(* CoDeSys 2.3.9.47 project: 2floor_2016-05-20.pr6 *)
(* Author: Yurko Shybaigolova *)
(* Libraries: TcAdsBC.lb6 5.7.02 11:03:02, standard.lb6 5.6.98 11:03:02, PlcSystemBC.lb6 21.3.01 11:03:02, TcPlcUtilitiesBC.lb6 13.5.05 11:19:40, TcBABasicBC.lb6 22.7.15 15:46:36 *)

(* Global variable list: main *)
VAR_GLOBAL
(*ADS*)
	ads_adr1: STRING:='10.0.5.61.1.1';
	ads_adr2: STRING:='10.0.5.62.1.1';
	ads_adr3: STRING:='10.0.5.63.1.1';

	write_ads: ADSWRITE;
	close_ads:ADSCLOSE;
	read_ads1: ADSREADEX;
	read_ads3: ADSREADEX;

	data1floor: ARRAY[0..4] OF BYTE;
	data1floor_prev: ARRAY[0..4] OF BYTE;
	data3floor: ARRAY[0..200] OF BYTE;
	data3floor_prev: ARRAY[0..200] OF BYTE;

	m_fancoil_kabinet_low 	AT%MX300.0: BOOL;
	m_fancoil_kabinet_med 	AT%MX300.1: BOOL;
	m_fancoil_kabinet_high 	AT%MX300.2: BOOL;
	m_fancoil_kino_low 		AT%MX300.3: BOOL;
	m_fancoil_kino_med 	AT%MX300.4: BOOL;
	m_fancoil_kino_high		AT%MX300.5: BOOL;

	tepla_pidloga_kabinet	AT%MX301.0:BOOL;
	tepla_pidloga_studio		AT%MX301.1:BOOL;

	m_klapan_kabinet		AT%MW302: WORD;


	m_klapan_kino			AT%MW304: WORD;

	sw_tambur3_2			AT%MX306.0:BOOL;
	bDarkOutside			AT%MX306.1:BOOL;
	bT_out_sign				AT%MX306.7:BOOL;

	eib_kabinet_shtory			AT%MX307.0:BOOL;
	eib_kabinet_tul				AT%MX307.1:BOOL;
	t_out3					AT%MB308:BYTE;
	t_out:REAL;
	iHour					AT%MB309:BYTE;
	iMinute					AT%MB310:BYTE;
	lights					AT%MB312:DWORD;

	eib_kino_shtory_move			AT%MX316.0:BOOL;
	eib_kino_tul_move				AT%MX316.1:BOOL;
	eib_kabinet_shtory_move		AT%MX316.2:BOOL;
	eib_kabinet_tul_move			AT%MX316.3:BOOL;
	eib_kino_shtory_position			AT%MB317	:BYTE;
	eib_kino_tul_position				AT%MB318	:BYTE;
	eib_kabinet_shtory_position		AT%MB319	:BYTE;
	eib_kabinet_tul_position			AT%MB320	:BYTE;


	eib_balkon_peryla 				AT%MX400.0:BOOL;
	eib_kino_l						AT%MX400.1:BOOL;
	eib_balkon_bra					AT%MX400.2:BOOL;
	eib_kabinet_balkon_l			AT%MX400.3:BOOL;
	eib_balkon						AT%MX400.4:BOOL;
	eib_korydor1					AT%MX400.5:BOOL;
	eib_kino_bra					AT%MX400.6:BOOL;
(*	eib_korydor2					AT%MX400.7:BOOL;
*)	eib_studio_pidsvitka				AT%MX401.0:BOOL;
	eib_skhody2_3					AT%MX401.1:BOOL;
	eib_studio_l						AT%MX401.2:BOOL;
(*	eib_kabinet_pidsvitka_kolo		AT%MX401.3:BOOL;
*)	eib_kabinet_svitlo				AT%MX401.4:BOOL;
	eib_kabinet_kobra				AT%MX401.5:BOOL;
	eib_tambur_l					AT%MX401.6:BOOL;
	eib_stend						AT%MX401.7:BOOL;
	eib_skhody_peryla				AT%MX402.0:BOOL;




	sw_tambur1_2			AT%MX100.0:BOOL;
	sw_vhid2				AT%MX100.1:BOOL;
	moove_kino				AT%MX101.0:BOOL;
	moove_skhody1_2		AT%MX101.1:BOOL;
	moove_studio			AT%MX101.2:BOOL;
	moove_kabinet			AT%MX101.3:BOOL;
	sw_tambur1_3_long		AT%MX101.4:BOOL;


	fbKino1_sw: FB_ShortLongClick;		(*processor for left button of the switch near the door in home cinema *)
END_VAR

(* Global variable list: physical *)
VAR_GLOBAL
(*	din1_1	AT %IX52.0:	BOOL;
	din1_2	AT %IX52.1:	BOOL;
	din1_3	AT %IX52.2:	BOOL;
	din1_4	AT %IX52.3:	BOOL;
	din1_5	AT %IX52.4:	BOOL;
	din1_6	AT %IX52.5:	BOOL;
	din1_7	AT %IX52.6:	BOOL;
	din1_8	AT %IX52.7:	BOOL;
	din2_1	AT %IX53.0:	BOOL;
	din2_2	AT %IX53.1:	BOOL;
	din2_3	AT %IX53.2:	BOOL;
	din2_4	AT %IX53.3:	BOOL;
	din2_5	AT %IX53.4:	BOOL;
	din2_6	AT %IX53.5:	BOOL;
	din2_7	AT %IX53.6:	BOOL;
	din2_8	AT %IX53.7:	BOOL;
*)

	sw_kino_balkon				AT %IX54.0:	BOOL;
	sw_tambur2_1				AT %IX54.1:	BOOL;
	sw_kino1					AT %IX54.2:	BOOL;
	sw_korydor					AT %IX54.3:	BOOL;
	sw_kino2					AT %IX54.4:	BOOL;
	sw_studio1					AT %IX54.5:	BOOL;
	sw_tambur2_2				AT %IX54.6:	BOOL;
	sw_studio2					AT %IX54.7:	BOOL;
	sw_kabinet1				AT %IX55.0:	BOOL;
(*	din4_2	AT %IX55.1:	BOOL;
*)	sw_kabinet2				AT %IX55.2:	BOOL;
	sw_kabinet2_1				AT %IX55.3:	BOOL;
	sw_kabinet_balkon			AT %IX55.4:	BOOL;
	sw_kabinet2_2				AT %IX55.5:	BOOL;
	sw_tambur3					AT %IX55.6:	BOOL;
(*	din4_8	AT %IX55.7:	BOOL;
*)

	balkon_peryla				AT %QX52.0:	BOOL;
	kino_l						AT %QX52.1:	BOOL;
	balkon_bra					AT %QX52.2:	BOOL;
	kabinet_balkon_l			AT %QX52.3:	BOOL;
	balkon						AT %QX52.4:	BOOL;
	korydor1					AT %QX52.5:	BOOL;
	kino_bra					AT %QX52.6:	BOOL;
	korydor2					AT %QX52.7:	BOOL;
	studio_pidsvitka 				AT %QX53.0:	BOOL;
	skhody2_3					AT %QX53.1:	BOOL;
	studio_l						AT %QX53.2:	BOOL;
	kabinet_pidsvitka_kolo		AT %QX53.3:	BOOL;
	kabinet_svitlo				AT %QX53.4:	BOOL;
	kabinet_kobra 				AT %QX53.5:	BOOL;
	tambur_l					AT %QX53.6:	BOOL;
	stend						AT %QX53.7:	BOOL;
	collector_kabinet1			AT %QX54.0:	BOOL;
	fancoil_kabinet_low			AT %QX54.1:	BOOL;
	collector_kabinet2			AT %QX54.2:	BOOL;
	fancoil_kabinet_med			AT %QX54.3:	BOOL;
	collector_studio1			AT %QX54.4:	BOOL;
	fancoil_kabinet_high			AT %QX54.5:	BOOL;
	collector_studio2			AT %QX54.6:	BOOL;
	fancoil_kino_low				AT %QX54.7:	BOOL;
	fancoil_kino_med			AT %QX55.0:	BOOL;
(*	dout4_2	AT %QX55.1:	BOOL;
*)	fancoil_kino_high			AT %QX55.2:	BOOL;
	skhody_peryla				AT %QX55.3:	BOOL;
(*	dout4_5	AT %QX55.4:	BOOL;
	dout4_6	AT %QX55.5:	BOOL;
	dout4_7	AT %QX55.6:	BOOL;
	dout4_8	AT %QX55.7:	BOOL;
*)	kino_tul_open				AT %QX56.0:	BOOL;
	kabinet_tul_close 			AT %QX56.1:	BOOL;
	kino_tul_close 				AT %QX56.2:	BOOL;
	kabinet_tul_open			AT %QX56.3:	BOOL;
	kino_shtory_open			AT %QX56.4:	BOOL;
	kabinet_shtory_open			AT %QX56.5:	BOOL;
	kino_shtory_close			AT %QX56.6:	BOOL;
	kabinet_shtory_close		AT %QX56.7:	BOOL;


	klapan_kino 				AT %QB2:	INT;
	klapan_kabinet				AT %QB6:	INT; (*0-opened, 16#7fff - closed*)

	temp_kabinet				AT %IB18:	INT;
	temp_studio		 			AT %IB26:	INT;


	Term_12_KL3228_4_1_State			AT %IB16:	USINT;

	Term_12_KL3228_4_1_Ctrl				AT %QB16:	USINT;
	Term_12_KL3228_4_1_Data_Out		AT %QB18:	INT;
	Term_12_KL3228_4_2_State			AT %IB20:	USINT;
	Term_12_KL3228_4_2_Data_In			AT %IB22:	INT;
	Term_12_KL3228_4_2_Ctrl				AT %QB20:	USINT;
	Term_12_KL3228_4_2_Data_Out		AT %QB22:	INT;
	Term_12_KL3228_4_3_State			AT %IB24:	USINT;

	Term_12_KL3228_4_3_Ctrl				AT %QB24:	USINT;
	Term_12_KL3228_4_3_Data_Out		AT %QB26:	INT;
	Term_12_KL3228_4_4_State			AT %IB28:	USINT;
	Term_12_KL3228_4_4_Data_In			AT %IB30:	INT;
	Term_12_KL3228_4_4_Ctrl				AT %QB28:	USINT;
	Term_12_KL3228_4_4_Data_Out		AT %QB30:	INT;
	Term_13_KL3228_4_1_State			AT %IB32:	USINT;
	Term_13_KL3228_4_1_Data_In			AT %IB34:	INT;
	Term_13_KL3228_4_1_Ctrl				AT %QB32:	USINT;
	Term_13_KL3228_4_1_Data_Out		AT %QB34:	INT;
	Term_13_KL3228_4_2_State			AT %IB36:	USINT;
	Term_13_KL3228_4_2_Data_In			AT %IB38:	INT;
	Term_13_KL3228_4_2_Ctrl				AT %QB36:	USINT;
	Term_13_KL3228_4_2_Data_Out		AT %QB38:	INT;
	Term_13_KL3228_4_3_State			AT %IB40:	USINT;
	Term_13_KL3228_4_3_Data_In			AT %IB42:	INT;
	Term_13_KL3228_4_3_Ctrl				AT %QB40:	USINT;
	Term_13_KL3228_4_3_Data_Out		AT %QB42:	INT;
	Term_13_KL3228_4_4_State			AT %IB44:	USINT;
	Term_13_KL3228_4_4_Data_In			AT %IB46:	INT;
	Term_13_KL3228_4_4_Ctrl				AT %QB44:	USINT;
	Term_13_KL3228_4_4_Data_Out		AT %QB46:	INT;
	Term_14_KL2761_State					AT %IB48:	USINT;
	kino_bra_state							AT %IB50:	INT;
	Term_14_KL2761_Ctrl					AT %QB48:	USINT;
	kino_bra_ctrl							AT %QB50:	INT;



END_VAR

(* POU MAIN, ST *)
PROGRAM MAIN
VAR

END_VAR
Light;
heat;
ADS1_write;
ADS3_write;
ADS_Communication;
END_PROGRAM

(* POU Light, CFC *)
PROGRAM Light
VAR
	longPressDelay: TIME:=t#500ms;
	lightDuration:INT:=120;




	fbKino_l							: FB_Light;						(*fb for home cinema mainlight switching*)
	fbKino_bra						: FB_Dimmer1SwitchEco;		(*fb for home cinema bra dimming*)
	fbKino2_sw						: FB_ShortLongClick;			(*processor for right button of the switch near the door in home cinema *)
	fbKino_bra_switching			: FB_Light;						(*fb for generating ON and OFF signals for 2SwitchDimmer fb*)
	fbKabinet_balkon				: FB_Light;		(*fb for balkony light switching in Oleg's cabinet*)
	fbKino_balkon					: FB_Light;		(*fb for switching balcony light in home cinema
			*)
	fbKabinet_l						: FB_Light;		(*fb for kabinet main light switching*)
	fbKabinet_kobra					: FB_Light;		(*fb for kabinet "cobra light" switching*)
	fStudio_l						: FB_Light;		(*fb for studio main light switching*)
	fStudio_pidsvitka				: FB_Light;		(*fb for studio  secondary light switching*)
	fbKorydor_l						: FB_Light;		(*fb for corridor light switching *)
	fbStend							: FB_Light;		(*fb for climbing wall light switching*)
	fbSkhody2_3					: FB_Light;		(*fb for stairs to the 3rd floor light switching*)

	fbKabinet1_sw: FB_ShortLongClick;				(*processor for left button of the kabinet switch near the door*)
	fbKabinet2_sw: FB_ShortLongClick;				(*processor for right button of the kabinet switch near the door*)
	fbKabinetShtory: FB_VenetianBlindEx1Switch;		(*fb for shtory control in kabinet*)

	fbKabinetShtorySwitching: FB_Light;				(*fb for ON and OFF signals generation for shtory control*)

	fbKabinetTulSwitching: FB_Light;					(*fb for ON and OFF signals generation for tul control*)
	fbKabinetTul: FB_VenetianBlindEx1Switch;		(*fb for ON and OFF signals generation for tul control*)

	fbKinoShtory: FB_VenetianBlindEx1Switch;
	kino_shtory_up_trigger: R_TRIG;
	kino_shtory_down_trigger: R_TRIG;

	kino_shtoryActualPosition: 	USINT;				(*position of the kino shtory*)
	kabinet_tulActualPosition: 	USINT;				(*position of the kabinet tul*)
	kabinet_shtoryActualPosition: USINT;				(*position of the kabinet shtory*)
	kino_tulActualPosition: 		USINT;					(*position of the kabinet shtory*)

	fbKinoTul: FB_VenetianBlindEx1Switch;
END_VAR
VAR CONSTANT
	msecMultiplier: DINT := 1000;
END_VAR
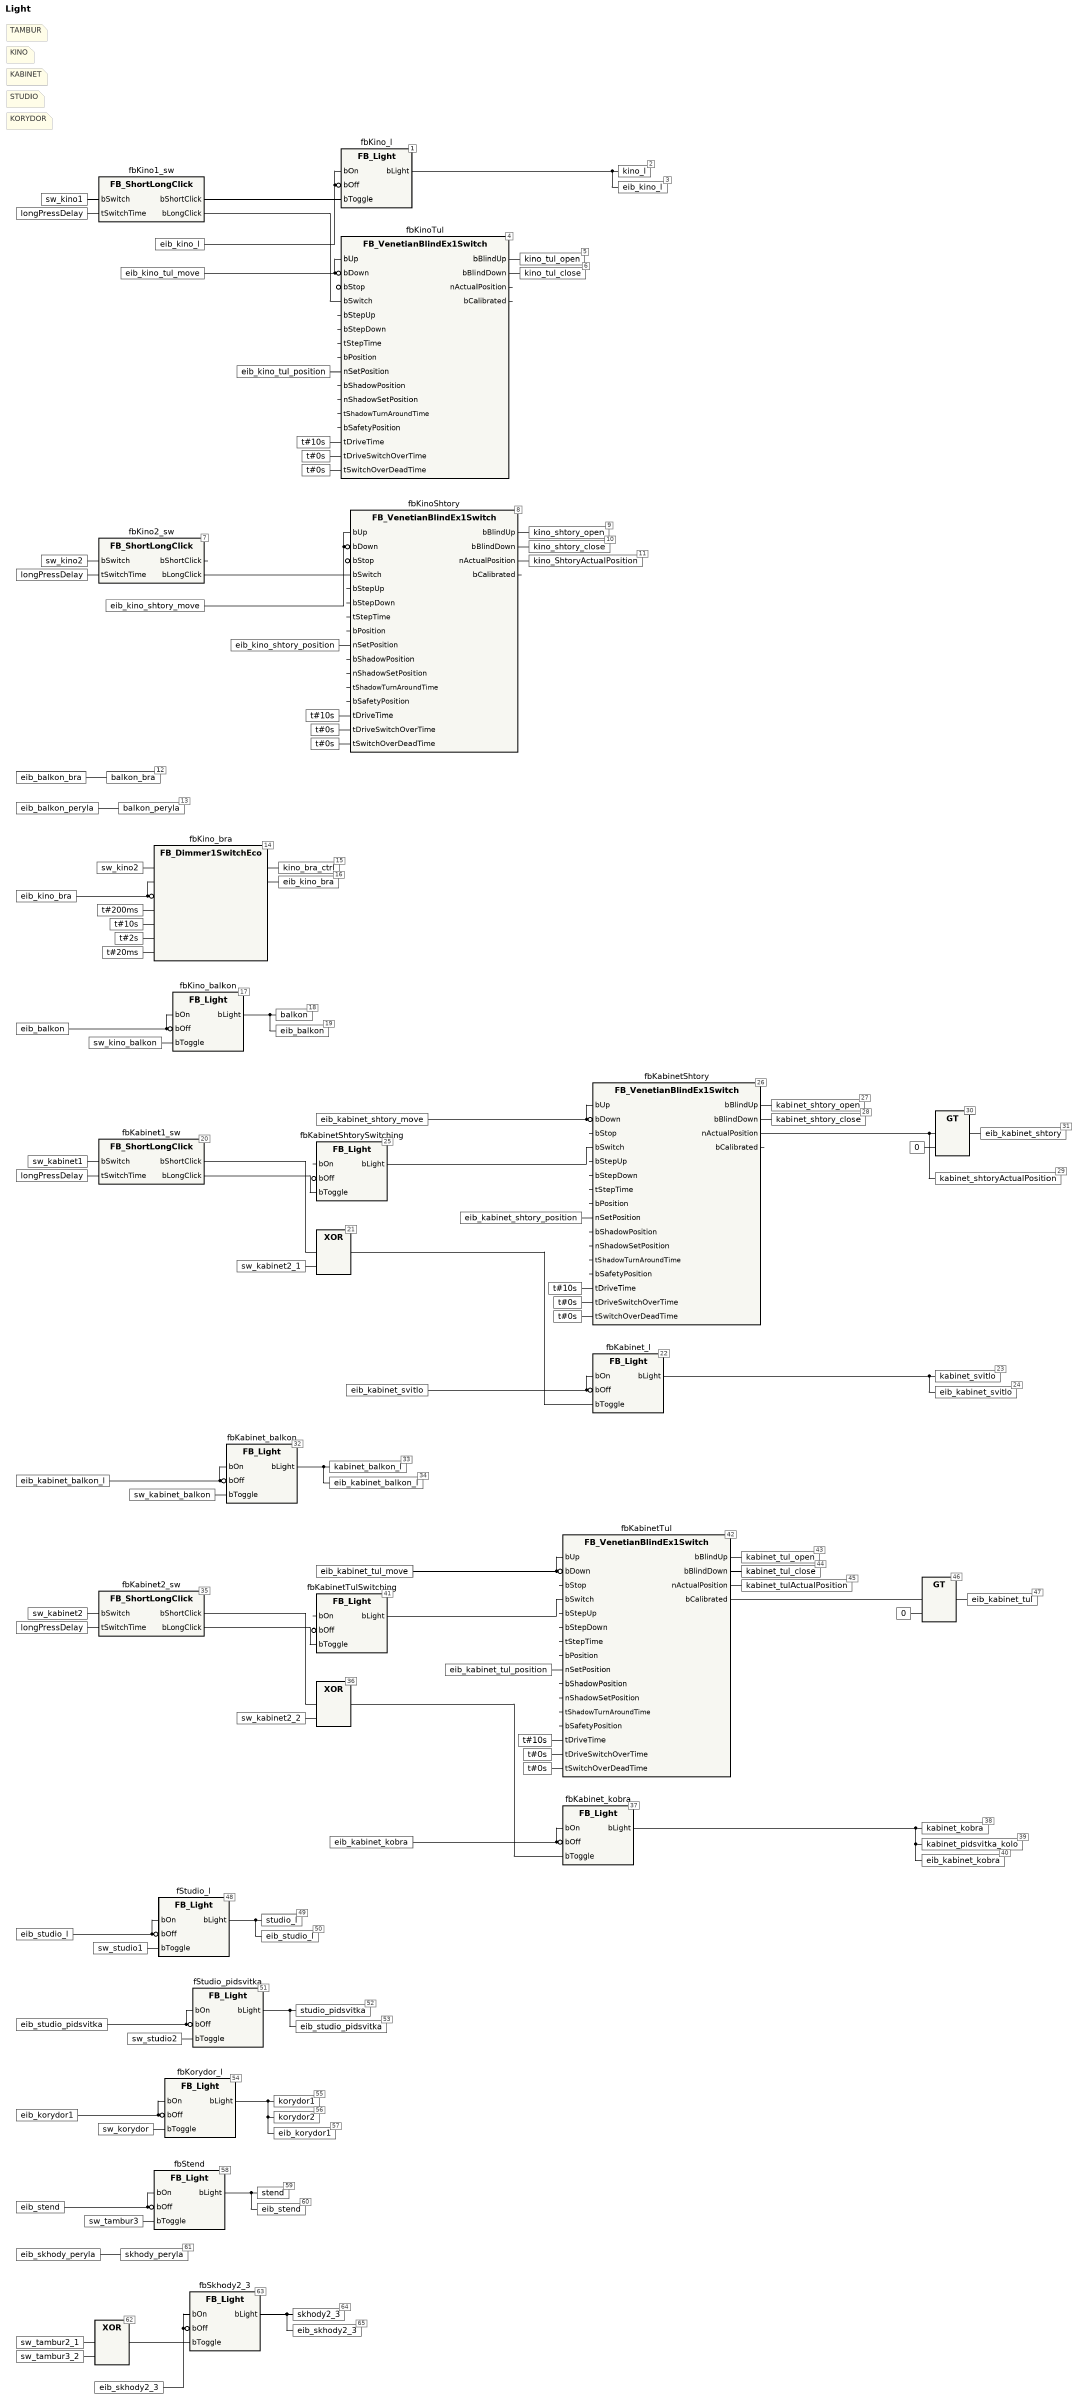
_CFC_ (* Continuous Function Chart, elements in execution order *)
(* TAMBUR *)
(* KINO *)
(* KABINET *)
(* STUDIO *)
(* KORYDOR *)
#0 fbKino1_sw:FB_ShortLongClick(bSwitch: sw_kino1, tSwitchTime: longPressDelay)
#1 fbKino_l:FB_Light(bOn: eib_kino_l, bOff: NOT eib_kino_l, bToggle: #0.bShortClick)
#2 kino_l <= #1.bLight
#3 eib_kino_l <= #1.bLight
#4 fbKinoTul:FB_VenetianBlindEx1Switch(bUp: eib_kino_tul_move, bDown: NOT eib_kino_tul_move, bStop: -, bSwitch: #0.bLongClick, bStepUp: -, bStepDown: -, tStepTime: -, bPosition: -, nSetPosition: eib_kino_tul_position, bShadowPosition: -, nShadowSetPosition: -, tShadowTurnAroundTime: -, bSafetyPosition: -, tDriveTime: t#10s, tDriveSwitchOverTime: t#0s, tSwitchOverDeadTime: t#0s)
#5 kino_tul_open <= #4.bBlindUp
#6 kino_tul_close <= #4.bBlindDown
#7 fbKino2_sw:FB_ShortLongClick(bSwitch: sw_kino2, tSwitchTime: longPressDelay)
#8 fbKinoShtory:FB_VenetianBlindEx1Switch(bUp: eib_kino_shtory_move, bDown: NOT eib_kino_shtory_move, bStop: -, bSwitch: #7.bLongClick, bStepUp: -, bStepDown: -, tStepTime: -, bPosition: -, nSetPosition: eib_kino_shtory_position, bShadowPosition: -, nShadowSetPosition: -, tShadowTurnAroundTime: -, bSafetyPosition: -, tDriveTime: t#10s, tDriveSwitchOverTime: t#0s, tSwitchOverDeadTime: t#0s)
#9 kino_shtory_open <= #8.bBlindUp
#10 kino_shtory_close <= #8.bBlindDown
#11 kino_ShtoryActualPosition <= #8.nActualPosition
#12 balkon_bra <= eib_balkon_bra
#13 balkon_peryla <= eib_balkon_peryla
#14 fbKino_bra:FB_Dimmer1SwitchEco(sw_kino2, eib_kino_bra, NOT eib_kino_bra, t#200ms, t#10s, t#2s, t#20ms)
#15 kino_bra_ctrl <= #14.out 1
#16 eib_kino_bra <= #14.out 2
#17 fbKino_balkon:FB_Light(bOn: eib_balkon, bOff: NOT eib_balkon, bToggle: sw_kino_balkon)
#18 balkon <= #17.bLight
#19 eib_balkon <= #17.bLight
#20 fbKabinet1_sw:FB_ShortLongClick(bSwitch: sw_kabinet1, tSwitchTime: longPressDelay)
#21 XOR(#20.bShortClick, sw_kabinet2_1)
#22 fbKabinet_l:FB_Light(bOn: eib_kabinet_svitlo, bOff: NOT eib_kabinet_svitlo, bToggle: #21)
#23 kabinet_svitlo <= #22.bLight
#24 eib_kabinet_svitlo <= #22.bLight
#25 fbKabinetShtorySwitching:FB_Light(bOn: -, bOff: -, bToggle: #20.bLongClick)
#26 fbKabinetShtory:FB_VenetianBlindEx1Switch(bUp: eib_kabinet_shtory_move, bDown: NOT eib_kabinet_shtory_move, bStop: -, bSwitch: #25.bLight, bStepUp: -, bStepDown: -, tStepTime: -, bPosition: -, nSetPosition: eib_kabinet_shtory_position, bShadowPosition: -, nShadowSetPosition: -, tShadowTurnAroundTime: -, bSafetyPosition: -, tDriveTime: t#10s, tDriveSwitchOverTime: t#0s, tSwitchOverDeadTime: t#0s)
#27 kabinet_shtory_open <= #26.bBlindUp
#28 kabinet_shtory_close <= #26.bBlindDown
#29 kabinet_shtoryActualPosition <= #26.nActualPosition
#30 GT(#26.nActualPosition, 0)
#31 eib_kabinet_shtory <= #30
#32 fbKabinet_balkon:FB_Light(bOn: eib_kabinet_balkon_l, bOff: NOT eib_kabinet_balkon_l, bToggle: sw_kabinet_balkon)
#33 kabinet_balkon_l <= #32.bLight
#34 eib_kabinet_balkon_l <= #32.bLight
#35 fbKabinet2_sw:FB_ShortLongClick(bSwitch: sw_kabinet2, tSwitchTime: longPressDelay)
#36 XOR(#35.bShortClick, sw_kabinet2_2)
#37 fbKabinet_kobra:FB_Light(bOn: eib_kabinet_kobra, bOff: NOT eib_kabinet_kobra, bToggle: #36)
#38 kabinet_kobra <= #37.bLight
#39 kabinet_pidsvitka_kolo <= #37.bLight
#40 eib_kabinet_kobra <= #37.bLight
#41 fbKabinetTulSwitching:FB_Light(bOn: -, bOff: -, bToggle: #35.bLongClick)
#42 fbKabinetTul:FB_VenetianBlindEx1Switch(bUp: eib_kabinet_tul_move, bDown: NOT eib_kabinet_tul_move, bStop: -, bSwitch: #41.bLight, bStepUp: -, bStepDown: -, tStepTime: -, bPosition: -, nSetPosition: eib_kabinet_tul_position, bShadowPosition: -, nShadowSetPosition: -, tShadowTurnAroundTime: -, bSafetyPosition: -, tDriveTime: t#10s, tDriveSwitchOverTime: t#0s, tSwitchOverDeadTime: t#0s)
#43 kabinet_tul_open <= #42.bBlindUp
#44 kabinet_tul_close <= #42.bBlindDown
#45 kabinet_tulActualPosition <= #42.nActualPosition
#46 GT(#42.bCalibrated, 0)
#47 eib_kabinet_tul <= #46
#48 fStudio_l:FB_Light(bOn: eib_studio_l, bOff: NOT eib_studio_l, bToggle: sw_studio1)
#49 studio_l <= #48.bLight
#50 eib_studio_l <= #48.bLight
#51 fStudio_pidsvitka:FB_Light(bOn: eib_studio_pidsvitka, bOff: NOT eib_studio_pidsvitka, bToggle: sw_studio2)
#52 studio_pidsvitka <= #51.bLight
#53 eib_studio_pidsvitka <= #51.bLight
#54 fbKorydor_l:FB_Light(bOn: eib_korydor1, bOff: NOT eib_korydor1, bToggle: sw_korydor)
#55 korydor1 <= #54.bLight
#56 korydor2 <= #54.bLight
#57 eib_korydor1 <= #54.bLight
#58 fbStend:FB_Light(bOn: eib_stend, bOff: NOT eib_stend, bToggle: sw_tambur3)
#59 stend <= #58.bLight
#60 eib_stend <= #58.bLight
#61 skhody_peryla <= eib_skhody_peryla
#62 XOR(sw_tambur2_1, sw_tambur3_2)
#63 fbSkhody2_3:FB_Light(bOn: eib_skhody2_3, bOff: NOT eib_skhody2_3, bToggle: #62)
#64 skhody2_3 <= #63.bLight
#65 eib_skhody2_3 <= #63.bLight
_END_CFC_
END_PROGRAM

(* POU heat, ST *)
PROGRAM heat
VAR
	fancoil_kino: WORD;
	fancoil_kabinet:  WORD;

	temp_measure: TOF;
	t_kabinet: REAL;
	t_studio: REAL;
	t_max: SINT;
	t_min: SINT;
	delta_kabinet: REAL;
	delta_studio:REAL;
	t_kabinetPrev: REAL;
	t_studioPrev: REAL;
	t_kabinet_sum: REAL;
	t_studio_sum: REAL;
	i: INT;
	retry: BOOL:=TRUE;		(*переміряти температуру*)
	iRetryCounter: INT;
END_VAR
	fancoil_kino_low:=m_fancoil_kino_low;
	fancoil_kino_med:=m_fancoil_kino_med;
	fancoil_kino_high:=m_fancoil_kino_high;
	klapan_kino:=m_klapan_kino;

	fancoil_kabinet_low:=m_fancoil_kabinet_low;
	fancoil_kabinet_med:=m_fancoil_kabinet_med;
	fancoil_kabinet_high:=m_fancoil_kabinet_high;
	klapan_kabinet:=m_klapan_kabinet;
IF bT_out_sign THEN t_out:=0-t_out3; ELSE t_out:=t_out3; END_IF;

(*фільтр показань сенсорів температури*)
CASE i OF
0..500: init;
ELSE
	IF retry THEN
		temp_measure.PT:=t#2s;
	ELSE
		temp_measure.PT:=t#5m;
	END_IF
	IF retry THEN
		IF iRetryCounter >5 THEN iRetryCounter:=0; i:=0; ELSE iRetryCounter:=iRetryCounter+1; END_IF;
	END_IF;
	temp_measure( IN:=NOT temp_measure.q); (*перевіряти температуру кожні 20 хв*)

IF NOT temp_measure.Q THEN

	delta_kabinet:=ABS(t_kabinetPrev-temp_kabinet*0.01);
	delta_studio:=ABS(t_studioPrev-temp_studio*0.01);
	retry:=FALSE;
	IF delta_kabinet<1 THEN
		t_kabinet:= temp_kabinet ;
	ELSE
		t_kabinet:=t_kabinetPrev;
		retry:=TRUE;
	END_IF

	IF delta_studio<1 THEN
		t_studio:= temp_studio ;
	ELSE
		t_studio:=t_studioPrev;
		retry:=TRUE;
	END_IF

	t_kabinetPrev:=t_kabinet;
	t_studioPrev:=t_studio;

END_IF
END_CASE



IF t_out>8 THEN
	t_max:=40;
	t_min:=10;
ELSE
	IF t_out >0 THEN
		t_max:=50;
	ELSE
		t_max:=70;
	END_IF
END_IF


	IF t_kabinet >= t_max THEN
		collector_kabinet1:=FALSE;
		collector_kabinet2:=FALSE;
	ELSE
		IF t_kabinet < t_min THEN
			collector_kabinet1:=TRUE;
			collector_kabinet2:=TRUE;
		ELSE
			collector_kabinet1:=tepla_pidloga_kabinet;
			collector_kabinet2:=tepla_pidloga_kabinet;
		END_IF
	END_IF


	IF t_studio >= t_max THEN
		collector_studio1:=FALSE;
		collector_studio2:=FALSE;
	ELSE
		IF t_studio < t_min THEN
			collector_studio1:=TRUE;
			collector_studio2:=TRUE;
		ELSE
			collector_studio1:=tepla_pidloga_studio;
			collector_studio2:=tepla_pidloga_studio;
		END_IF
	END_IF
END_PROGRAM
ACTION init:
IF i=500 THEN
	t_kabinetPrev:=t_kabinet_sum/i;
	t_studioPrev:=t_studio_sum/i;
	t_studio_sum:=0;
	t_kabinet_sum:=0;
	i:=501;
ELSE
	t_kabinet_sum:=t_kabinet_sum+temp_kabinet*0.01;
	t_studio_sum:=t_studio_sum+temp_studio*0.01;
	i:=i+1;
END_IF
END_ACTION

(* POU ADS1_write, ST *)
PROGRAM ADS1_write
VAR
	write_timeout: TIME;
	b_write1: BOOL;
	write_ads1: ADSWRITE;

	timer1:TP;
	errorcounter1, pack_c:CTU ;
	test_word: WORD;
	i1,j1: INT;
	data_changed: BOOL;
	try_again1: BOOL;
END_VAR
data1floor[0].0:=sw_tambur2_2;

(*1floor*)
FOR i1:=0 TO (SIZEOF(data1floor))-1 DO
	IF data1floor[i1]<>data1floor_prev[i1] THEN
		b_write1:=TRUE;
		EXIT;
	ELSE
		b_write1:=FALSE;
	END_IF
END_FOR

IF try_again1 AND NOT timer1.Q THEN
	b_write1:=TRUE;
	try_again1:=FALSE;
END_IF

(*

IF write_ads1.BUSY THEN b_write1:=FALSE; END_IF

	write_ads1(
		NETID:=ads_adr1,
		PORT:=800,
		IDXGRP:=16#4020,
		IDXOFFS:=200,
		WRITE:=b_write1,
		TMOUT:=t#5s,
		LEN:=SIZEOF(data1floor),
		SRCADDR:=ADR(data1floor));

IF write_ads1.ERR AND NOT timer1.Q THEN
	timer1.IN:=TRUE;
	try_again1:=TRUE;
END_IF
timer1(PT:=write_timeout);
timer1.IN:=FALSE;
*)

FOR j1:=0 TO (SIZEOF(data1floor))-1 DO
	data1floor_prev[j1]:=data1floor[j1];
END_FOR
END_PROGRAM

(* POU ADS3_write, ST *)
PROGRAM ADS3_write
VAR
	write_timeout: TIME;
	b_write1: BOOL;
	write_ads1: ADSWRITE;

	timer1:TP;
	errorcounter1:CTU ;
	test_word: WORD;
	i1,j1: INT;
	data_changed: BOOL;
	try_again1: BOOL;
END_VAR
VAR CONSTANT
	fb_heartbeat_timer: TON;
END_VAR
data3floor[0].0:=balkon_peryla;
data3floor[0].1:=kino_l;
data3floor[0].2:=balkon_bra;
data3floor[0].3:=kabinet_balkon_l;
data3floor[0].4:=balkon;
data3floor[0].5:=korydor1;
data3floor[0].6:=kino_bra;
data3floor[0].7:=korydor2;
data3floor[1].0:=studio_pidsvitka;
data3floor[1].1:=skhody2_3;
data3floor[1].2:=studio_l;
data3floor[1].3:=kabinet_pidsvitka_kolo;
data3floor[1].4:=kabinet_svitlo;
data3floor[1].5:=kabinet_kobra;
data3floor[1].6:=tambur_l;
data3floor[1].7:=stend;
data3floor[2].0:=skhody_peryla;


data3floor[3].0:=collector_kabinet1;
data3floor[3].1:=collector_kabinet2;
data3floor[3].2:=collector_studio1;
data3floor[3].3:=collector_studio2;

data3floor[3].4:=fancoil_kabinet_low;
data3floor[3].5:=fancoil_kabinet_med;
data3floor[3].6:=fancoil_kabinet_high;

data3floor[3].7:=fancoil_kino_low;
data3floor[4].0:=fancoil_kino_med;
data3floor[4].1:=fancoil_kino_high;


data3floor[5]:=Light.kabinet_shtoryActualPosition;
data3floor[6]:=Light.kabinet_tulActualPosition;
data3floor[7]:=Light.kino_shtoryActualPosition;
data3floor[8]:=Light.kino_tulActualPosition;



fb_heartbeat_timer(in:=NOT fb_heartbeat_timer.Q, pt:=t#10s);
(*3floor*)
data_changed:=FALSE;
FOR i1:=0 TO (SIZEOF(data3floor))-1 DO
	IF data3floor[i1]<>data3floor_prev[i1]  OR try_again1 THEN
		b_write1:=TRUE;
		data_changed:=TRUE;
		EXIT;
	ELSE
		b_write1:=FALSE;
	END_IF
END_FOR

(*
IF write_ads1.BUSY THEN b_write1:=FALSE; END_IF

	write_ads1(
		NETID:=ads_adr3,
		PORT:=800,
		IDXGRP:=16#4020,
		IDXOFFS:=200,
		WRITE:=b_write1,
		TMOUT:=t#300ms,
		LEN:=SIZEOF(data3floor),
		SRCADDR:=ADR(data3floor));


write_ads1.WRITE:=FALSE;
errorcounter1(cu:=write_ads1.ERR);
IF write_ads1.ERR AND NOT timer1.Q THEN
	timer1.IN:=TRUE;
	try_again1:=TRUE;
ELSE try_again1:=FALSE;
END_IF
timer1(PT:=write_timeout*2);
timer1.IN:=FALSE;
*)


FOR j1:=0 TO (SIZEOF(data3floor))-1 DO
	data3floor_prev[j1]:=data3floor[j1];
END_FOR
END_PROGRAM

(* POU ADS_Communication, CFC *)
PROGRAM ADS_Communication
VAR

	fb_floor1ADSwrite: ADSWRITE;
	fb_floor3ADSwrite: ADSWRITE;
END_VAR
VAR (* helpers for the ST form of the networks *)
	_t10 : DWORD;
	_t21 : DWORD;
	_t23 : DWORD;
END_VAR
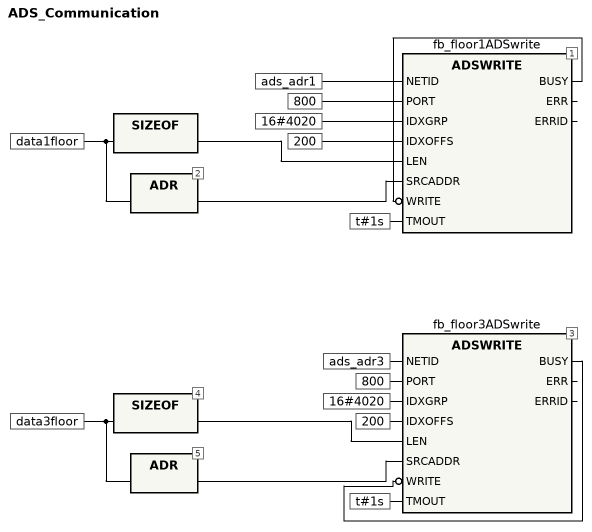
_CFC_ (* Continuous Function Chart, elements in execution order *)
#0 SIZEOF(data1floor)
#1 fb_floor1ADSwrite:ADSWRITE(NETID: ads_adr1, PORT: 800, IDXGRP: 16#4020, IDXOFFS: 200, LEN: #0, SRCADDR: #2, WRITE: NOT #1.BUSY, TMOUT: t#1s)
#2 ADR(data1floor)
#3 fb_floor3ADSwrite:ADSWRITE(NETID: ads_adr3, PORT: 800, IDXGRP: 16#4020, IDXOFFS: 200, LEN: #4, SRCADDR: #5, WRITE: NOT #3.BUSY, TMOUT: t#1s)
#4 SIZEOF(data3floor)
#5 ADR(data3floor)
_END_CFC_
(* the same logic as Structured Text *)
fb_floor1ADSwrite(NETID := ads_adr1, PORT := 800, IDXGRP := 16#4020, IDXOFFS := 200, LEN := SIZEOF(data1floor), SRCADDR := _t10, WRITE := NOT fb_floor1ADSwrite.BUSY, TMOUT := t#1s);
_t10 := ADR(data1floor);
fb_floor3ADSwrite(NETID := ads_adr3, PORT := 800, IDXGRP := 16#4020, IDXOFFS := 200, LEN := _t21, SRCADDR := _t23, WRITE := NOT fb_floor3ADSwrite.BUSY, TMOUT := t#1s);
_t21 := SIZEOF(data3floor);
_t23 := ADR(data3floor);
END_PROGRAM

(* POU light_old, ST *)
PROGRAM light_old
VAR
	kino_balkon, kino1, kino2, studio1,studio2, kabinet1, kabinet2, kabinet_balkon, korydor, tambur1, tambur2, tambur3: SWITCH;
	switch_delay: TIME;
	off_delay: TIME;
	fbDarkEdge, fbTambur3_2:R_TRIG;

	prev_eib_balkon_peryla 		:BOOL;
	prev_eib_kino_l				:BOOL;
	prev_eib_balkon_bra			:BOOL;
	prev_eib_kabinet_balkon_l		:BOOL;
	prev_eib_balkon				:BOOL;
	prev_eib_korydor1			:BOOL;
	prev_eib_kino_bra			:BOOL;
	prev_eib_korydor2			:BOOL;
	prev_eib_studio_pidsvitka		:BOOL;
	prev_eib_skhody2_3			:BOOL;
	prev_eib_studio_l				:BOOL;
	prev_eib_kabinet_pidsvitka_kolo :BOOL;
	prev_eib_kabinet_svitlo		:BOOL;
	prev_eib_kabinet_kobra		:BOOL;
	prev_eib_tambur_l				:BOOL;
	prev_eib_stend				:BOOL;
	prev_eib_skhody_peryla		:BOOL;
	fb_kino_l_f_edge:F_TRIG;

END_VAR
switch_delay:=t#500ms; (*затримка довгого натискання*)
off_delay:=t#3m; (*затримка для відкладеного вимкнення*)

kino_balkon(MODE:='short&long', IN:=sw_kino_balkon,SWITCH_DELAY:=switch_delay, Q_SHORT=>balkon );

fb_kino_l_f_edge(CLk:=eib_kino_l);
IF eib_kino_l =  prev_eib_kino_l THEN
	kino1(MODE:='short&long',IN:=sw_kino1, SWITCH_DELAY:=switch_delay);
	IF kino1.short THEN kino_l:= NOT kino_l; END_IF
	eib_kino_l:=kino_l;
ELSE
	kino_l:=eib_kino_l;
END_IF
prev_eib_kino_l:=eib_kino_l;

IF eib_kino_bra = prev_eib_kino_bra THEN
	kino2(MODE:='short&long', IN:=sw_kino2, SWITCH_DELAY:=switch_delay);
	IF kino2.short THEN kino_bra:= NOT kino_bra; END_IF
	eib_kino_bra:=kino_bra;
ELSE kino_bra:=eib_kino_bra;
END_IF
prev_eib_kino_bra:=eib_kino_bra;

IF eib_studio_l = eib_studio_l THEN
	studio1(MODE:='short&long', IN:=sw_studio1, SWITCH_DELAY:=switch_delay);
	IF studio1.short THEN studio_l := NOT studio_l; END_IF;
	eib_studio_l:=studio_l;
ELSE
	studio_l:=eib_studio_l;
END_IF
prev_eib_studio_l:=eib_studio_l;

IF eib_studio_pidsvitka= prev_eib_studio_pidsvitka THEN
	studio2(MODE:='short&long', IN:=sw_studio2, SWITCH_DELAY:=switch_delay);
	IF studio2.short THEN studio_pidsvitka:= NOT studio_pidsvitka; END_IF
	eib_studio_pidsvitka:=studio_pidsvitka;
ELSE
	studio_pidsvitka:=eib_studio_pidsvitka;
END_IF
prev_eib_studio_pidsvitka:=eib_studio_pidsvitka;

IF (eib_korydor1 = prev_eib_korydor1) THEN
	korydor(MODE:='short&long', IN:=sw_korydor, SWITCH_DELAY:=switch_delay);
	IF korydor.short THEN korydor1:= NOT korydor1;END_IF
	eib_korydor1:=korydor1;
ELSE
	IF eib_korydor1 XOR prev_eib_korydor1 THEN  korydor1:=eib_korydor1;END_IF
END_IF
korydor2:=korydor1;
prev_eib_korydor1:=eib_korydor1;


kabinet1(MODE:='short&long', IN:=sw_kabinet1 XOR sw_kabinet2_1, SWITCH_DELAY:=switch_delay);
IF eib_kabinet_svitlo = prev_eib_kabinet_svitlo THEN
	IF kabinet1.short THEN kabinet_svitlo:= NOT kabinet_svitlo; END_IF;
	eib_kabinet_svitlo:=kabinet_svitlo;
ELSE
	kabinet_svitlo:=eib_kabinet_svitlo;
END_IF
	prev_eib_kabinet_svitlo:=eib_kabinet_svitlo;

kabinet2(MODE:='short&long', IN:=sw_kabinet2 XOR sw_kabinet2_2, SWITCH_DELAY:=switch_delay);
IF (eib_kabinet_kobra = prev_eib_kabinet_kobra) OR (eib_kabinet_pidsvitka_kolo = 	prev_eib_kabinet_pidsvitka_kolo) THEN
	IF kabinet2.short THEN
		IF NOT (kabinet_kobra OR kabinet_pidsvitka_kolo) THEN
			kabinet_kobra:=TRUE; kabinet_pidsvitka_kolo:=TRUE;
		ELSE
			 kabinet_kobra:=FALSE; kabinet_pidsvitka_kolo:=FALSE;
		END_IF;
		eib_kabinet_kobra:=kabinet_kobra;
		eib_kabinet_pidsvitka_kolo:=kabinet_pidsvitka_kolo;
	END_IF
END_IF

IF eib_kabinet_kobra <> prev_eib_kabinet_kobra THEN kabinet_kobra:=eib_kabinet_kobra; END_IF;
prev_eib_kabinet_kobra:=eib_kabinet_kobra;
IF eib_kabinet_pidsvitka_kolo <> prev_eib_kabinet_pidsvitka_kolo THEN kabinet_pidsvitka_kolo:=eib_kabinet_pidsvitka_kolo; END_IF;
prev_eib_kabinet_pidsvitka_kolo:=eib_kabinet_pidsvitka_kolo;

kabinet_balkon(MODE:='short&long', IN:=sw_kabinet_balkon, SWITCH_DELAY:=switch_delay);
IF eib_kabinet_balkon_l= prev_eib_kabinet_balkon_l THEN
	IF kabinet_balkon.short THEN kabinet_balkon_l:= NOT kabinet_balkon_l; END_IF;
	eib_kabinet_balkon_l:=kabinet_balkon_l;
ELSE
	kabinet_balkon_l:=eib_kabinet_balkon_l;
END_IF
prev_eib_kabinet_balkon_l:=eib_kabinet_balkon_l;
fbTambur3_2(CLK:=sw_tambur3_2);
sw_tambur3_2:=FALSE;
tambur1(MODE:='light', IN:=sw_tambur2_1 OR fbTambur3_2.Q , SWITCH_DELAY:=switch_delay);
tambur2(MODE:='light', IN:=sw_tambur2_2 OR sw_tambur1_2 , SWITCH_DELAY:=switch_delay);
tambur3(MODE:='short&long', IN:=sw_tambur3 OR sw_vhid2, SWITCH_DELAY:=switch_delay);

IF eib_stend = prev_eib_stend THEN
	IF tambur3.short THEN stend:= NOT stend; END_IF;
	eib_stend:=stend;
ELSE
	stend:=eib_stend;
END_IF
prev_eib_stend:=eib_stend;

IF eib_skhody2_3 = prev_eib_skhody2_3 THEN
	IF tambur1.short THEN skhody2_3:=NOT skhody2_3; END_IF
	eib_skhody2_3:=skhody2_3;
ELSE
	skhody2_3:=eib_skhody2_3;
END_IF
prev_eib_skhody2_3:=eib_skhody2_3;

fbDarkEdge(CLK:=bDarkOutside);

IF (eib_skhody_peryla = prev_eib_skhody_peryla) OR  (eib_balkon_bra = prev_eib_balkon_bra) OR (eib_balkon_peryla = prev_eib_balkon_bra)THEN
	IF fbDarkEdge.Q AND iHour>16  THEN
		skhody_peryla:=TRUE;
		balkon_bra:=TRUE;
		balkon_peryla:=TRUE;
	END_IF

	IF ihour=00 AND iminute=00THEN
		skhody_peryla:=FALSE;
		balkon_bra:=FALSE;
		balkon_peryla:=FALSE;
	END_IF
		eib_skhody_peryla:=skhody_peryla;
		eib_balkon_bra:=balkon_bra;
		eib_balkon_peryla:=balkon_peryla;
END_IF

IF eib_skhody_peryla <> prev_eib_skhody_peryla THEN skhody_peryla:=eib_skhody_peryla;END_IF
prev_eib_skhody_peryla:=eib_skhody_peryla;
IF eib_balkon_bra<>prev_eib_balkon_bra THEN  balkon_bra:=eib_balkon_bra;END_IF
prev_eib_balkon_bra:=eib_balkon_bra;
IF eib_balkon_peryla <> prev_eib_balkon_peryla  THEN balkon_peryla:=eib_balkon_peryla;END_IF
prev_eib_balkon_peryla:=eib_balkon_peryla;
END_PROGRAM

(* POU Vymykachi/SWITCH, ST *)
FUNCTION_BLOCK SWITCH
VAR_INPUT
	IN:BOOL;
	SWITCH_DELAY:TIME; (*різниця між коротким і довгим натисненням*)
	SHORT_OFF_DELAY, LONG_OFF_DELAY: TIME; (*час затримки вимкнення по короткому та довгому натисненню*)
	MODE:STRING; (*delayed, light, light&vent, short&long, delayed_short&long, *)
	NUMBER_OF_OUTS:INT;
END_VAR
VAR_OUTPUT
	Q_SHORT:BOOL:=FALSE;
	Q_SHORT_D: BOOL;(*вихід для вимкнення із затримкою, вмикається разом із виходом короткого натискання*)
	Q_LONG:BOOL:=FALSE;
	Q_LONG_D:BOOL; (*вихід для вимкнення із затримкою, вмикається разом із виходом довгого натискання*)
END_VAR
VAR
	STAN:BOOL:=FALSE;
	Q_S_fall:F_TRIG; (*ловить задній фронт вихода короткого натискання*)
	Q_L_fall:F_TRIG;(*ловить задній фронт вихода довгого натискання*)
	chas: TIME; (*час доки кнопка натиснена*)

	long: BOOL; (*стає тру, якщо було довге натиснення*)
	short: BOOL; (*стає тру, якщо було коротке натиснення*)
	timer, short_off_delay_timer, long_off_delay_timer: TON; (*таймери: час натискання, час переключення відкладеного виходу по довгому та короткому натисканнях*)
	up: BOOL; (*кнопка натиснена*)

	delay_l, delay_s:BOOL; (*запускати таймери відкладеного вимкнення*)

	turn_off_long: BOOL;
	start_l, start_s:BOOL;
END_VAR
short:=0;
long:=0;
timer(IN:=IN AND STAN, PT:=t#10s);
IF IN AND STAN THEN
	chas:=timer.ET;
	up:=1;
ELSE
up:=0;
END_IF;

IF NOT IN AND NOT STAN THEN
chas:=t#0ms;
END_IF;

IF STAN AND NOT IN THEN
	IF chas <SWITCH_DELAY THEN
		short:=1;
		Q_SHORT:= NOT Q_SHORT;
	END_IF;
	IF chas>=SWITCH_DELAY THEN
		Q_LONG:= NOT Q_LONG;
		long:=1;
	END_IF;
END_IF;

(*затримка вимикання*)
Q_L_fall(CLK:=Q_LONG);
Q_S_fall(CLK:=Q_SHORT);

IF Q_L_FALL.Q THEN
		start_l:=TRUE;
END_IF

IF Q_S_FALL.Q THEN
	start_s:=TRUE;
END_IF

IF MODE='light&vent' THEN
	IF start_s THEN start_l:=start_s; END_IF
END_IF

IF LONG_OFF_DELAY <> t#0ms THEN (*виконувати лише якщо в блок переданий параметр затримки на вимкнення*)

	IF Q_LONG THEN
		Q_LONG_D:=Q_LONG;
	END_IF

	long_off_delay_timer(IN:=start_l, PT:=LONG_OFF_DELAY);

	IF long_off_delay_timer.Q THEN
		Q_LONG_D:=FALSE;
		start_l:=FALSE;
	END_IF

ELSE
	Q_LONG_D:=Q_LONG;
END_IF

IF SHORT_OFF_DELAY <> t#0ms THEN (*виконувати лише якщо в блок переданий параметр затримки на вимкнення*)

	IF Q_SHORT THEN
		Q_SHORT_D:=Q_SHORT;
	END_IF

	short_off_delay_timer(IN:=start_s, PT:=SHORT_OFF_DELAY);

	IF short_off_delay_timer.Q THEN
		Q_SHORT_D:=FALSE;
		start_s:=FALSE;
	END_IF


ELSE
	Q_SHORT_D:=Q_SHORT;
END_IF

IF MODE='delayed' THEN
	Q_LONG:=Q_LONG_D;
	Q_SHORT:=Q_SHORT_D;
END_IF
(*працють лише короткі замикання*)
IF MODE='light' THEN
	Q_SHORT_D:=FALSE;
	Q_LONG:=Q_SHORT;
	Q_LONG_D:=FALSE;
END_IF
(*затримки не працюють*)
IF MODE='short&long' THEN
	Q_SHORT_D:=FALSE;
	Q_LONG_D:=FALSE;
END_IF
(*при вимкненні всього світла вимикати вентилятор і затримкою*)
IF MODE='light&vent' THEN
	IF NOT Q_SHORT AND Q_LONG THEN
		Q_LONG:=Q_LONG_D;
	END_IF
END_IF

STAN := IN;
END_FUNCTION_BLOCK

(* POU shtory_kabinet_old, ST *)
PROGRAM shtory_kabinet_old
VAR
	inc1, inc: UINT;
	impulse: BOOL;
	shtory_status: BOOL; (*1 - closed, 0 - opened*)
	impulse1: BOOL;
	tul_status: BOOL; (*1 - closed, 0 - opened*)
	lift_move_dir, lift_moves: BOOL;
	rising1: BOOL;
	falling1: BOOL;
	rising2: BOOL;
	falling2: BOOL;
	inc2: UINT;
	panel_shtory_move, panel_tul_move :BOOL;

	(*таймери для формування керуючих імпульсів*)
	timer_shtory_move, timer_shtory_stop,timer_tul_move, timer_tul_stop, move_lift_up, move_lift_down: TP;

	shtory_counter, tul_counter, lift_counter: UINT;
	counter:CTU;

	shtory_move: BOOL;
	shtory_stop: BOOL;
	tul_move: BOOL;
	eib_tul_move: BOOL;
	eib_shtory_move: BOOL;
	R_SHTORY:R_TRIG;
	F_SHTORY:F_TRIG;
	R_TUL:R_TRIG;
	F_TUL:F_TRIG;

	bBlock: BOOL;
	darkness_shtory_move: TP;
END_VAR
bBlock:=FALSE;
kabinet_shtory_open:=FALSE;
kabinet_shtory_close:=FALSE;
kabinet_tul_open:=FALSE;
kabinet_tul_close:=FALSE;
IF iHour=9 AND iMinute=0  THEN
	bBlock:=TRUE;
	kabinet_shtory_open:=TRUE;
	kabinet_shtory_close:=FALSE;
END_IF

darkness_shtory_move(IN:=bDarkOutside, PT:=t#15s);
IF darkness_shtory_move.Q THEN
	kabinet_shtory_open:=FALSE;
	kabinet_shtory_close:=TRUE;
	kabinet_tul_open:=FALSE;
	kabinet_tul_close:=TRUE;
	bBlock:=TRUE;
END_IF

IF NOT bBlock THEN
(*детекція відсутності фронтів*)
IF Light.kabinet1.Q_LONG = impulse THEN
	rising1:=0;
	falling1:=0;
END_IF;

IF light.kabinet2.Q_LONG = impulse1 THEN
	rising2:=0;
	falling2:=0;
END_IF;

(*ловим передній фронт довгого натискання першої клавіші*)
IF light.kabinet1.Q_LONG AND NOT impulse  THEN
	rising1:=1;
	falling1:=0;
END_IF;

(*задній фронт*)
IF NOT light.kabinet1.Q_LONG AND  impulse THEN
	falling1:=1;
	rising1:=0;
END_IF;

(*ловим передній фронт довгого натискання другої клавіші*)
IF light.kabinet2.Q_LONG AND NOT impulse1  THEN
	rising2:=1;
	falling2:=0;
END_IF;

(*ловим задній фронт довгого натискання другої клавіші*)
IF NOT light.kabinet2.Q_LONG AND  impulse1 THEN
	falling2:=1;
	rising2:=0;
END_IF;


(*команди шторам смарт баса на 3 поверсі*)
R_SHTORY(CLK:=kabinet_shtory, Q=>eib_shtory_move);
IF NOT R_SHTORY.Q THEN F_SHTORY(CLK:=kabinet_shtory, Q=>eib_shtory_move); END_IF

R_TUL(CLK:=kabinet_tul, Q=>eib_tul_move);
IF NOT R_TUL.Q THEN F_TUL(CLK:=kabinet_tul, Q=>eib_tul_move); END_IF

shtory_move:= rising1 OR falling1 OR eib_shtory_move;
tul_move:= rising2 OR falling2 OR eib_tul_move;

(*формування імпульсів для керування шторами, тюлями та ліфтом*)
timer_shtory_move(IN:=shtory_move, PT:=t#1000ms);
timer_shtory_stop(IN:=shtory_move , PT:=t#1000ms);
timer_tul_move(IN:=tul_move  , PT:=t#1000ms);
timer_tul_stop(IN:=tul_move , PT:=t#1000ms);

	(*вибір рухати чи зупинити  штори*)
	IF shtory_move THEN
		inc:=inc+1;
	END_IF;
	IF inc>2 THEN inc:=1; END_IF;

	(*вибір рухати чи зупинити  тюль*)
	IF tul_move THEN
		inc1:=inc1+1;
	END_IF;
	IF inc1>2 THEN inc1:=1; END_IF;

	CASE inc OF

	1:
		kabinet_shtory_open:=timer_shtory_move.Q; (*відкривати*)
		kabinet_shtory_close:= 0;
		shtory_status:=1;

	2:
		kabinet_shtory_close:=timer_shtory_move.Q;(*закривати*)
		kabinet_shtory_open:= 0;
		shtory_status:=0;

	END_CASE;

	CASE inc1 OF

	1:
		kabinet_tul_open:=timer_tul_move.Q; (*відкривати*)
		kabinet_tul_close:= 0;
		tul_status:=1;
	2:
		kabinet_tul_close:=timer_tul_move.Q;(*закривати*)
		kabinet_tul_open:= 0;
		tul_status:=0;

	END_CASE;


(*запам'ятовування стану довгого натискання для детекції фронтів*)

impulse:=light.kabinet1.Q_LONG;
impulse1:=light.kabinet2.Q_LONG;
END_IF
END_PROGRAM

(* POU shtory_kino_old, ST *)
PROGRAM shtory_kino_old
VAR
	inc1, inc: UINT;
	impulse: BOOL;
	shtory_status: BOOL;(*1 - closed, 0 - opened*)
	impulse1: BOOL;
	tul_status: BOOL;(*1 - closed, 0 - opened*)
	lift_move_dir, lift_moves: BOOL;
	rising1: BOOL;
	falling1: BOOL;
	rising2: BOOL;
	falling2: BOOL;
	inc2: UINT;
	panel_shtory_move, panel_tul_move :BOOL;
	(*таймери для формування керуючих імпульсів*)
	timer_shtory_move, timer_shtory_stop,timer_tul_move, timer_tul_stop, move_lift_up, move_lift_down: TP;

	shtory_counter, tul_counter, lift_counter: UINT;
	counter:CTU;

	shtory_move: BOOL;
	shtory_stop: BOOL;
	tul_move: BOOL;
	eib_tul_move: BOOL;
	eib_shtory_move: BOOL;
	R_SHTORY:R_TRIG;
	F_SHTORY:F_TRIG;
	R_TUL:R_TRIG;
	F_TUL:F_TRIG;

END_VAR
(*детекція відсутності фронтів*)
IF light.kino1.Q_LONG = impulse THEN
	rising1:=0;
	falling1:=0;
END_IF;

IF light.kino2.Q_LONG = impulse1 THEN
	rising2:=0;
	falling2:=0;
END_IF;

(*ловим передній фронт довгого натискання першої клавіші*)
IF light.kino1.Q_LONG AND NOT impulse  THEN
	rising1:=1;
	falling1:=0;
END_IF;

(*задній фронт*)
IF NOT Light.kino1.Q_LONG AND  impulse THEN
	falling1:=1;
	rising1:=0;
END_IF;

(*ловим передній фронт довгого натискання другої клавіші*)
IF light.kino2.Q_LONG AND NOT impulse1  THEN
	rising2:=1;
	falling2:=0;
END_IF;

(*ловим задній фронт довгого натискання другої клавіші*)
IF NOT light.kino2.Q_LONG AND  impulse1 THEN
	falling2:=1;
	rising2:=0;
END_IF;


(*команди шторам смарт баса на 3 поверсі*)
R_SHTORY(CLK:=kino_shtory, Q=>eib_shtory_move);
IF NOT R_SHTORY.Q THEN F_SHTORY(CLK:=kino_shtory, Q=>eib_shtory_move); END_IF

R_TUL(CLK:=kino_tul, Q=>eib_tul_move);
IF NOT R_TUL.Q THEN F_TUL(CLK:=kino_tul, Q=>eib_tul_move); END_IF


shtory_move:= rising1 OR falling1 OR eib_shtory_move;
tul_move:= rising2 OR falling2 OR eib_tul_move;

(*формування імпульсів для керування шторами, тюлями та ліфтом*)
timer_shtory_move(IN:=shtory_move, PT:=t#1500ms);
timer_shtory_stop(IN:=shtory_move , PT:=t#1500ms);
timer_tul_move(IN:=tul_move  , PT:=t#1500ms);
timer_tul_stop(IN:=tul_move , PT:=t#1500ms);

	(*вибір рухати чи зупинити  штори*)
	IF shtory_move THEN
		inc:=inc+1;
	END_IF;
	IF inc>2 THEN inc:=1; END_IF;

	(*вибір рухати чи зупинити  тюль*)
	IF tul_move THEN
		inc1:=inc1+1;
	END_IF;
	IF inc1>2 THEN inc1:=1; END_IF;

	CASE inc OF

	1:
		kino_shtory_open:=timer_shtory_move.Q; (*відкривати*)
		kino_shtory_close:= 0;
		shtory_status:=1;

	2:
		kino_shtory_close:=timer_shtory_move.Q;(*закривати*)
		kino_shtory_open:= 0;
		shtory_status:=0;

	END_CASE;

	CASE inc1 OF

	1:
		kino_tul_open:=timer_tul_move.Q; (*відкривати*)
		kino_tul_close:= 0;
		tul_status:=1;
	2:
		kino_tul_close:=timer_tul_move.Q;(*закривати*)
		kino_tul_open:= 0;
		tul_status:=0;

	END_CASE;


(*запам'ятовування стану довгого натискання для детекції фронтів*)

impulse:=light.kino1.Q_LONG;
impulse1:=light.kino2.Q_LONG;
END_PROGRAM
